{attribute 'qualified_only'}
TYPE ENUM_TM2K4_States :
(
    // Adapted from ENUM_ATM_States to add TARGET6

    Unknown := 0,
    OUT := 1,
    TARGET1 := 2,
    TARGET2 := 3,
    TARGET3 := 4,
    YAG := 5,
    DIODE := 6
) UINT;
END_TYPE

(* stored: Version 1.1.0.1, ProductVersion 3.1.4024.12
   DUT ENUM_TM2K4_States: Id {f3c92633-68cb-466f-8e8c-2fc04f05fc6a} *)
